TYPE DistanceSensorConfigs :
STRUCT
	MicroEpsilonDistanceSensorConfig : MicroEpsilonDistanceSensorConfig;
END_STRUCT
END_TYPE

(* stored: Version 1.1.0.1, ProductVersion 3.1.4024.12
   DUT DistanceSensorConfigs: Id {870858f1-a187-436f-91f9-3101c4b9e1b2} *)
